    movel([0.144923, -1.275155, -2.596829, -0.840405, 1.570796, 1.715720],accel_mss,speed_ms,0,blend_radius_m)
    movel([0.144342, -1.274168, -2.597401, -0.840819, 1.570796, 1.715139],accel_mss,speed_ms,0,blend_radius_m)
    movel([0.143423, -1.273257, -2.597929, -0.841203, 1.570796, 1.714219],accel_mss,speed_ms,0,blend_radius_m)
    movel([0.142097, -1.272464, -2.598387, -0.841538, 1.570796, 1.712893],accel_mss,speed_ms,0,blend_radius_m)
    movel([0.140296, -1.271830, -2.598753, -0.841806, 1.570796, 1.711092],accel_mss,speed_ms,0,blend_radius_m)
    # Splitting Linear movement in 4 (instruction 536: MoveL 457)
    movel([0.138191, -1.271393, -2.599005, -0.841991, 1.570796, 1.708987],accel_mss,speed_ms,0,blend_radius_m)
    movel([0.136082, -1.270961, -2.599254, -0.842174, 1.570796, 1.706878],accel_mss,speed_ms,0,blend_radius_m)
    movel([0.133968, -1.270534, -2.599499, -0.842356, 1.570796, 1.704764],accel_mss,speed_ms,0,blend_radius_m)
    movel([0.131850, -1.270113, -2.599741, -0.842535, 1.570796, 1.702647],accel_mss,speed_ms,0,blend_radius_m)
    # Splitting Linear movement in 6 (instruction 537: MoveL 458)
    movel([0.129903, -1.269748, -2.599951, -0.842690, 1.570796, 1.700700],accel_mss,speed_ms,0,blend_radius_m)
    movel([0.127953, -1.269388, -2.600157, -0.842843, 1.570796, 1.698749],accel_mss,speed_ms,0,blend_radius_m)
    movel([0.125999, -1.269032, -2.600361, -0.842995, 1.570796, 1.696795],accel_mss,speed_ms,0,blend_radius_m)
    movel([0.124041, -1.268681, -2.600563, -0.843145, 1.570796, 1.694838],accel_mss,speed_ms,0,blend_radius_m)
    movel([0.122081, -1.268335, -2.600761, -0.843293, 1.570796, 1.692877],accel_mss,speed_ms,0,blend_radius_m)
    movel([0.120116, -1.267993, -2.600957, -0.843439, 1.570796, 1.690913],accel_mss,speed_ms,0,blend_radius_m)
    speed_ms = 0.005
    # Splitting Linear movement in 4 (instruction 539: MoveL 459)
    movel([0.120116, -1.265890, -2.599818, -0.846681, 1.570796, 1.690913],accel_mss,speed_ms,0,blend_radius_m)
    movel([0.120116, -1.263799, -2.598675, -0.849915, 1.570796, 1.690913],accel_mss,speed_ms,0,blend_radius_m)
    movel([0.120116, -1.261719, -2.597530, -0.853140, 1.570796, 1.690913],accel_mss,speed_ms,0,blend_radius_m)
    movel([0.120116, -1.259651, -2.596381, -0.856357, 1.570796, 1.690913],accel_mss,speed_ms,0,blend_radius_m)
    speed_ms = 0.040
    # Splitting Linear movement in 12 (instruction 541: MoveL 460)
    movel([0.118639, -1.261858, -2.595130, -0.855401, 1.570796, 1.689436],accel_mss,speed_ms,0,blend_radius_m)
    movel([0.117169, -1.264057, -2.593878, -0.854454, 1.570796, 1.687965],accel_mss,speed_ms,0,blend_radius_m)
    movel([0.115705, -1.266250, -2.592623, -0.853516, 1.570796, 1.686501],accel_mss,speed_ms,0,blend_radius_m)
    movel([0.114247, -1.268435, -2.591368, -0.852586, 1.570796, 1.685043],accel_mss,speed_ms,0,blend_radius_m)
    movel([0.112796, -1.270613, -2.590110, -0.851666, 1.570796, 1.683592],accel_mss,speed_ms,0,blend_radius_m)
    movel([0.111350, -1.272785, -2.588851, -0.850753, 1.570796, 1.682147],accel_mss,speed_ms,0,blend_radius_m)
    movel([0.109912, -1.274949, -2.587590, -0.849850, 1.570796, 1.680708],accel_mss,speed_ms,0,blend_radius_m)
    movel([0.108479, -1.277107, -2.586327, -0.848955, 1.570796, 1.679275],accel_mss,speed_ms,0,blend_radius_m)
    movel([0.107053, -1.279258, -2.585063, -0.848068, 1.570796, 1.677849],accel_mss,speed_ms,0,blend_radius_m)
    movel([0.105632, -1.281402, -2.583797, -0.847190, 1.570796, 1.676429],accel_mss,speed_ms,0,blend_radius_m)
    movel([0.104218, -1.283539, -2.582530, -0.846320, 1.570796, 1.675014],accel_mss,speed_ms,0,blend_radius_m)
    movel([0.102810, -1.285670, -2.581261, -0.845458, 1.570796, 1.673606],accel_mss,speed_ms,0,blend_radius_m)
    speed_ms = 0.005
    # Splitting Linear movement in 4 (instruction 543: MoveL 461)
    movel([0.102810, -1.287713, -2.582382, -0.842294, 1.570796, 1.673606],accel_mss,speed_ms,0,blend_radius_m)
    movel([0.102810, -1.289767, -2.583499, -0.839123, 1.570796, 1.673606],accel_mss,speed_ms,0,blend_radius_m)
    movel([0.102810, -1.291832, -2.584614, -0.835943, 1.570796, 1.673606],accel_mss,speed_ms,0,blend_radius_m)
    movel([0.102810, -1.293908, -2.585724, -0.832757, 1.570796, 1.673606],accel_mss,speed_ms,0,blend_radius_m)
    speed_ms = 0.035
    # Splitting Linear movement in 4 (instruction 545: MoveL 462)
    movel([0.104961, -1.293243, -2.586126, -0.833020, 1.570796, 1.675758],accel_mss,speed_ms,0,blend_radius_m)
    movel([0.107114, -1.292580, -2.586525, -0.833284, 1.570796, 1.677910],accel_mss,speed_ms,0,blend_radius_m)
    movel([0.109268, -1.291921, -2.586922, -0.833546, 1.570796, 1.680064],accel_mss,speed_ms,0,blend_radius_m)
    movel([0.111423, -1.291264, -2.587316, -0.833808, 1.570796, 1.682219],accel_mss,speed_ms,0,blend_radius_m)
    speed_ms = 0.005
    # Splitting Linear movement in 6 (instruction 547: MoveL 463)
    movel([0.111423, -1.289877, -2.586574, -0.835938, 1.570796, 1.682219],accel_mss,speed_ms,0,blend_radius_m)
    movel([0.111423, -1.288495, -2.585831, -0.838063, 1.570796, 1.682219],accel_mss,speed_ms,0,blend_radius_m)
    movel([0.111423, -1.287118, -2.585085, -0.840186, 1.570796, 1.682219],accel_mss,speed_ms,0,blend_radius_m)
    movel([0.111423, -1.285745, -2.584339, -0.842305, 1.570796, 1.682219],accel_mss,speed_ms,0,blend_radius_m)
    movel([0.111423, -1.284378, -2.583591, -0.844421, 1.570796, 1.682219],accel_mss,speed_ms,0,blend_radius_m)
    movel([0.111423, -1.283015, -2.582841, -0.846533, 1.570796, 1.682219],accel_mss,speed_ms,0,blend_radius_m)
    speed_ms = 0.040
    # Splitting Linear movement in 6 (instruction 549: MoveL 464)
    movel([0.113420, -1.282408, -2.583201, -0.846780, 1.570796, 1.684216],accel_mss,speed_ms,0,blend_radius_m)
    movel([0.115418, -1.281804, -2.583559, -0.847026, 1.570796, 1.686214],accel_mss,speed_ms,0,blend_radius_m)
    movel([0.117416, -1.281203, -2.583915, -0.847271, 1.570796, 1.688213],accel_mss,speed_ms,0,blend_radius_m)
    movel([0.119416, -1.280604, -2.584269, -0.847516, 1.570796, 1.690212],accel_mss,speed_ms,0,blend_radius_m)
    movel([0.121417, -1.280007, -2.584621, -0.847761, 1.570796, 1.692213],accel_mss,speed_ms,0,blend_radius_m)
    movel([0.123418, -1.279413, -2.584971, -0.848004, 1.570796, 1.694214],accel_mss,speed_ms,0,blend_radius_m)
    speed_ms = 0.005
    # Splitting Linear movement in 6 (instruction 551: MoveL 465)
    movel([0.123418, -1.280778, -2.585724, -0.845887, 1.570796, 1.694214],accel_mss,speed_ms,0,blend_radius_m)
    movel([0.123418, -1.282148, -2.586474, -0.843766, 1.570796, 1.694214],accel_mss,speed_ms,0,blend_radius_m)
    movel([0.123418, -1.283523, -2.587224, -0.841642, 1.570796, 1.694214],accel_mss,speed_ms,0,blend_radius_m)
    movel([0.123418, -1.284903, -2.587971, -0.839515, 1.570796, 1.694214],accel_mss,speed_ms,0,blend_radius_m)
    movel([0.123418, -1.286288, -2.588717, -0.837384, 1.570796, 1.694214],accel_mss,speed_ms,0,blend_radius_m)
    movel([0.123418, -1.287678, -2.589462, -0.835249, 1.570796, 1.694214],accel_mss,speed_ms,0,blend_radius_m)
    speed_ms = 0.035
    # Splitting Linear movement in 4 (instruction 553: MoveL 466)
    movel([0.125386, -1.287119, -2.589795, -0.835475, 1.570796, 1.696182],accel_mss,speed_ms,0,blend_radius_m)
    movel([0.127354, -1.286563, -2.590126, -0.835700, 1.570796, 1.698151],accel_mss,speed_ms,0,blend_radius_m)
    movel([0.129323, -1.286009, -2.590455, -0.835925, 1.570796, 1.700120],accel_mss,speed_ms,0,blend_radius_m)
    movel([0.131293, -1.285459, -2.590782, -0.836149, 1.570796, 1.702090],accel_mss,speed_ms,0,blend_radius_m)
    movel([0.133014, -1.284863, -2.591135, -0.836391, 1.570796, 1.703811],accel_mss,speed_ms,0,blend_radius_m)
    movel([0.134155, -1.284224, -2.591513, -0.836652, 1.570796, 1.704951],accel_mss,speed_ms,0,blend_radius_m)
    movel([0.135046, -1.283460, -2.591965, -0.836964, 1.570796, 1.705842],accel_mss,speed_ms,0,blend_radius_m)
    movel([0.135680, -1.282694, -2.592417, -0.837278, 1.570796, 1.706476],accel_mss,speed_ms,0,blend_radius_m)
    movel([0.136054, -1.282045, -2.592800, -0.837544, 1.570796, 1.706850],accel_mss,speed_ms,0,blend_radius_m)
    movel([0.136254, -1.281407, -2.593175, -0.837807, 1.570796, 1.707050],accel_mss,speed_ms,0,blend_radius_m)
    movel([0.136336, -1.280413, -2.593759, -0.838217, 1.570796, 1.707133],accel_mss,speed_ms,0,blend_radius_m)
    movel([0.136227, -1.279892, -2.594065, -0.838432, 1.570796, 1.707023],accel_mss,speed_ms,0,blend_radius_m)
    movel([0.135967, -1.279413, -2.594346, -0.838630, 1.570796, 1.706763],accel_mss,speed_ms,0,blend_radius_m)
    movel([0.135513, -1.279021, -2.594575, -0.838792, 1.570796, 1.706310],accel_mss,speed_ms,0,blend_radius_m)
    movel([0.134824, -1.278762, -2.594727, -0.838900, 1.570796, 1.705620],accel_mss,speed_ms,0,blend_radius_m)
    # Splitting Linear movement in 6 (instruction 565: MoveL 478)
    movel([0.132749, -1.278413, -2.594931, -0.839045, 1.570796, 1.703546],accel_mss,speed_ms,0,blend_radius_m)
    movel([0.130671, -1.278069, -2.595132, -0.839188, 1.570796, 1.701467],accel_mss,speed_ms,0,blend_radius_m)
    movel([0.128589, -1.277730, -2.595330, -0.839329, 1.570796, 1.699385],accel_mss,speed_ms,0,blend_radius_m)
    movel([0.126503, -1.277396, -2.595525, -0.839468, 1.570796, 1.697299],accel_mss,speed_ms,0,blend_radius_m)
    movel([0.124413, -1.277068, -2.595716, -0.839605, 1.570796, 1.695210],accel_mss,speed_ms,0,blend_radius_m)
    movel([0.122320, -1.276744, -2.595905, -0.839740, 1.570796, 1.693117],accel_mss,speed_ms,0,blend_radius_m)
    # Splitting Linear movement in 8 (instruction 566: MoveL 479)
    movel([0.122076, -1.278708, -2.594758, -0.838922, 1.570796, 1.692872],accel_mss,speed_ms,0,blend_radius_m)
    movel([0.121832, -1.280667, -2.593610, -0.838112, 1.570796, 1.692628],accel_mss,speed_ms,0,blend_radius_m)
    movel([0.121589, -1.282620, -2.592461, -0.837308, 1.570796, 1.692386],accel_mss,speed_ms,0,blend_radius_m)
    movel([0.121348, -1.284567, -2.591310, -0.836512, 1.570796, 1.692144],accel_mss,speed_ms,0,blend_radius_m)
    movel([0.121107, -1.286509, -2.590158, -0.835722, 1.570796, 1.691903],accel_mss,speed_ms,0,blend_radius_m)
    movel([0.120868, -1.288446, -2.589004, -0.834939, 1.570796, 1.691664],accel_mss,speed_ms,0,blend_radius_m)
    movel([0.120629, -1.290377, -2.587849, -0.834163, 1.570796, 1.691426],accel_mss,speed_ms,0,blend_radius_m)
    movel([0.120392, -1.292303, -2.586692, -0.833394, 1.570796, 1.691188],accel_mss,speed_ms,0,blend_radius_m)
    speed_ms = 0.005
    # Splitting Linear movement in 4 (instruction 568: MoveL 480)
    movel([0.120392, -1.290225, -2.585579, -0.836584, 1.570796, 1.691188],accel_mss,speed_ms,0,blend_radius_m)
    movel([0.120392, -1.288159, -2.584463, -0.839767, 1.570796, 1.691188],accel_mss,speed_ms,0,blend_radius_m)
    movel([0.120392, -1.286103, -2.583344, -0.842942, 1.570796, 1.691188],accel_mss,speed_ms,0,blend_radius_m)
    movel([0.120392, -1.284058, -2.582221, -0.846110, 1.570796, 1.691188],accel_mss,speed_ms,0,blend_radius_m)
    speed_ms = 0.040
    # Splitting Linear movement in 12 (instruction 570: MoveL 481)
    movel([0.119907, -1.286179, -2.580956, -0.845253, 1.570796, 1.690703],accel_mss,speed_ms,0,blend_radius_m)
    movel([0.119424, -1.288294, -2.579690, -0.844405, 1.570796, 1.690220],accel_mss,speed_ms,0,blend_radius_m)
    movel([0.118943, -1.290401, -2.578422, -0.843565, 1.570796, 1.689739],accel_mss,speed_ms,0,blend_radius_m)
    movel([0.118465, -1.292503, -2.577153, -0.842733, 1.570796, 1.689261],accel_mss,speed_ms,0,blend_radius_m)
    movel([0.117988, -1.294598, -2.575882, -0.841909, 1.570796, 1.688785],accel_mss,speed_ms,0,blend_radius_m)
    movel([0.117514, -1.296686, -2.574609, -0.841093, 1.570796, 1.688311],accel_mss,speed_ms,0,blend_radius_m)
    movel([0.117042, -1.298768, -2.573335, -0.840285, 1.570796, 1.687839],accel_mss,speed_ms,0,blend_radius_m)
    movel([0.116573, -1.300844, -2.572060, -0.839485, 1.570796, 1.687369],accel_mss,speed_ms,0,blend_radius_m)
    movel([0.116105, -1.302914, -2.570782, -0.838693, 1.570796, 1.686901],accel_mss,speed_ms,0,blend_radius_m)
    movel([0.115640, -1.304977, -2.569504, -0.837908, 1.570796, 1.686436],accel_mss,speed_ms,0,blend_radius_m)
    movel([0.115176, -1.307034, -2.568224, -0.837131, 1.570796, 1.685973],accel_mss,speed_ms,0,blend_radius_m)
    movel([0.114715, -1.309085, -2.566942, -0.836362, 1.570796, 1.685512],accel_mss,speed_ms,0,blend_radius_m)
    speed_ms = 0.005
    # Splitting Linear movement in 6 (instruction 572: MoveL 482)
    movel([0.114715, -1.310429, -2.567673, -0.834287, 1.570796, 1.685512],accel_mss,speed_ms,0,blend_radius_m)
    movel([0.114715, -1.311778, -2.568403, -0.832208, 1.570796, 1.685512],accel_mss,speed_ms,0,blend_radius_m)
    movel([0.114715, -1.313131, -2.569131, -0.830127, 1.570796, 1.685512],accel_mss,speed_ms,0,blend_radius_m)
    movel([0.114715, -1.314489, -2.569857, -0.828042, 1.570796, 1.685512],accel_mss,speed_ms,0,blend_radius_m)
    movel([0.114715, -1.315852, -2.570582, -0.825955, 1.570796, 1.685512],accel_mss,speed_ms,0,blend_radius_m)
    movel([0.114715, -1.317219, -2.571306, -0.823864, 1.570796, 1.685512],accel_mss,speed_ms,0,blend_radius_m)
    speed_ms = 0.035
    movel([0.113872, -1.317605, -2.571061, -0.823723, 1.570796, 1.684668],accel_mss,speed_ms,0,blend_radius_m)
    movel([0.113052, -1.317884, -2.570884, -0.823621, 1.570796, 1.683848],accel_mss,speed_ms,0,blend_radius_m)
    movel([0.111543, -1.318120, -2.570734, -0.823534, 1.570796, 1.682339],accel_mss,speed_ms,0,blend_radius_m)
    movel([0.110880, -1.318079, -2.570761, -0.823550, 1.570796, 1.681676],accel_mss,speed_ms,0,blend_radius_m)
    movel([0.109799, -1.317678, -2.571015, -0.823696, 1.570796, 1.680595],accel_mss,speed_ms,0,blend_radius_m)
    movel([0.109406, -1.317320, -2.571242, -0.823827, 1.570796, 1.680202],accel_mss,speed_ms,0,blend_radius_m)
    movel([0.108993, -1.316375, -2.571840, -0.824174, 1.570796, 1.679790],accel_mss,speed_ms,0,blend_radius_m)
    movel([0.108987, -1.315364, -2.572479, -0.824546, 1.570796, 1.679783],accel_mss,speed_ms,0,blend_radius_m)
    movel([0.109341, -1.314017, -2.573327, -0.825045, 1.570796, 1.680137],accel_mss,speed_ms,0,blend_radius_m)
    movel([0.109909, -1.312888, -2.574037, -0.825464, 1.570796, 1.680705],accel_mss,speed_ms,0,blend_radius_m)
    movel([0.110621, -1.311896, -2.574659, -0.825834, 1.570796, 1.681417],accel_mss,speed_ms,0,blend_radius_m)
    movel([0.111393, -1.311055, -2.575186, -0.826148, 1.570796, 1.682189],accel_mss,speed_ms,0,blend_radius_m)
    movel([0.112144, -1.310376, -2.575611, -0.826403, 1.570796, 1.682940],accel_mss,speed_ms,0,blend_radius_m)
    movel([0.114992, -1.307950, -2.577122, -0.827317, 1.570796, 1.685788],accel_mss,speed_ms,0,blend_radius_m)
    movel([0.116059, -1.306889, -2.577780, -0.827719, 1.570796, 1.686856],accel_mss,speed_ms,0,blend_radius_m)
    movel([0.117029, -1.305645, -2.578551, -0.828193, 1.570796, 1.687826],accel_mss,speed_ms,0,blend_radius_m)
    movel([0.117834, -1.304414, -2.579312, -0.828663, 1.570796, 1.688630],accel_mss,speed_ms,0,blend_radius_m)
    movel([0.118394, -1.303386, -2.579945, -0.829058, 1.570796, 1.689190],accel_mss,speed_ms,0,blend_radius_m)
    movel([0.118876, -1.302219, -2.580663, -0.829507, 1.570796, 1.689672],accel_mss,speed_ms,0,blend_radius_m)
    movel([0.119170, -1.301159, -2.581313, -0.829917, 1.570796, 1.689966],accel_mss,speed_ms,0,blend_radius_m)
    movel([0.119460, -1.299307, -2.582446, -0.830636, 1.570796, 1.690257],accel_mss,speed_ms,0,blend_radius_m)
    speed_ms = 0.005
    # Splitting Linear movement in 6 (instruction 596: MoveL 504)
    movel([0.119460, -1.297926, -2.581710, -0.832753, 1.570796, 1.690257],accel_mss,speed_ms,0,blend_radius_m)
    movel([0.119460, -1.296550, -2.580972, -0.834867, 1.570796, 1.690257],accel_mss,speed_ms,0,blend_radius_m)
    movel([0.119460, -1.295178, -2.580233, -0.836978, 1.570796, 1.690257],accel_mss,speed_ms,0,blend_radius_m)
    movel([0.119460, -1.293811, -2.579492, -0.839086, 1.570796, 1.690257],accel_mss,speed_ms,0,blend_radius_m)
    movel([0.119460, -1.292450, -2.578749, -0.841190, 1.570796, 1.690257],accel_mss,speed_ms,0,blend_radius_m)
    movel([0.119460, -1.291092, -2.578005, -0.843291, 1.570796, 1.690257],accel_mss,speed_ms,0,blend_radius_m)
    speed_ms = 0.040
    # Splitting Linear movement in 4 (instruction 598: MoveL 505)
    movel([0.117830, -1.291504, -2.577757, -0.843128, 1.570796, 1.688627],accel_mss,speed_ms,0,blend_radius_m)
    movel([0.116201, -1.291917, -2.577507, -0.842965, 1.570796, 1.686997],accel_mss,speed_ms,0,blend_radius_m)
    movel([0.114572, -1.292332, -2.577256, -0.842801, 1.570796, 1.685368],accel_mss,speed_ms,0,blend_radius_m)
    movel([0.112943, -1.292749, -2.577004, -0.842636, 1.570796, 1.683739],accel_mss,speed_ms,0,blend_radius_m)
    speed_ms = 0.005
    # Splitting Linear movement in 6 (instruction 600: MoveL 506)
    movel([0.112943, -1.294105, -2.577746, -0.840537, 1.570796, 1.683739],accel_mss,speed_ms,0,blend_radius_m)
    movel([0.112943, -1.295466, -2.578488, -0.838435, 1.570796, 1.683739],accel_mss,speed_ms,0,blend_radius_m)
    movel([0.112943, -1.296831, -2.579227, -0.836330, 1.570796, 1.683739],accel_mss,speed_ms,0,blend_radius_m)
    movel([0.112943, -1.298202, -2.579965, -0.834222, 1.570796, 1.683739],accel_mss,speed_ms,0,blend_radius_m)
    movel([0.112943, -1.299577, -2.580702, -0.832110, 1.570796, 1.683739],accel_mss,speed_ms,0,blend_radius_m)
    movel([0.112943, -1.300957, -2.581437, -0.829995, 1.570796, 1.683739],accel_mss,speed_ms,0,blend_radius_m)
    speed_ms = 0.035
    movel([0.112634, -1.302487, -2.580498, -0.829404, 1.570796, 1.683431],accel_mss,speed_ms,0,blend_radius_m)
    movel([0.112220, -1.303581, -2.579825, -0.828983, 1.570796, 1.683016],accel_mss,speed_ms,0,blend_radius_m)
    movel([0.111539, -1.304692, -2.579140, -0.828557, 1.570796, 1.682335],accel_mss,speed_ms,0,blend_radius_m)
    movel([0.110449, -1.305905, -2.578390, -0.828094, 1.570796, 1.681246],accel_mss,speed_ms,0,blend_radius_m)
    movel([0.109369, -1.306856, -2.577801, -0.827732, 1.570796, 1.680165],accel_mss,speed_ms,0,blend_radius_m)
    movel([0.107828, -1.307928, -2.577136, -0.827326, 1.570796, 1.678624],accel_mss,speed_ms,0,blend_radius_m)
    speed_ms = 0.005
    # Splitting Linear movement in 6 (instruction 609: MoveL 513)
    movel([0.107828, -1.306553, -2.576405, -0.829430, 1.570796, 1.678624],accel_mss,speed_ms,0,blend_radius_m)
    movel([0.107828, -1.305184, -2.575674, -0.831532, 1.570796, 1.678624],accel_mss,speed_ms,0,blend_radius_m)
    movel([0.107828, -1.303819, -2.574940, -0.833630, 1.570796, 1.678624],accel_mss,speed_ms,0,blend_radius_m)
    movel([0.107828, -1.302458, -2.574206, -0.835725, 1.570796, 1.678624],accel_mss,speed_ms,0,blend_radius_m)
    movel([0.107828, -1.301103, -2.573470, -0.837817, 1.570796, 1.678624],accel_mss,speed_ms,0,blend_radius_m)
    movel([0.107828, -1.299752, -2.572732, -0.839906, 1.570796, 1.678624],accel_mss,speed_ms,0,blend_radius_m)
    speed_ms = 0.040
    # Splitting Linear movement in 6 (instruction 611: MoveL 514)
    movel([0.108730, -1.297552, -2.574080, -0.840757, 1.570796, 1.679526],accel_mss,speed_ms,0,blend_radius_m)
    movel([0.109636, -1.295346, -2.575427, -0.841616, 1.570796, 1.680432],accel_mss,speed_ms,0,blend_radius_m)
    movel([0.110546, -1.293132, -2.576772, -0.842485, 1.570796, 1.681343],accel_mss,speed_ms,0,blend_radius_m)
    movel([0.111461, -1.290911, -2.578115, -0.843363, 1.570796, 1.682257],accel_mss,speed_ms,0,blend_radius_m)
    movel([0.112380, -1.288682, -2.579457, -0.844250, 1.570796, 1.683176],accel_mss,speed_ms,0,blend_radius_m)
    movel([0.113304, -1.286446, -2.580797, -0.845146, 1.570796, 1.684100],accel_mss,speed_ms,0,blend_radius_m)
    speed_ms = 0.005
    # Splitting Linear movement in 4 (instruction 613: MoveL 515)
    movel([0.113304, -1.288488, -2.581917, -0.841984, 1.570796, 1.684100],accel_mss,speed_ms,0,blend_radius_m)
    movel([0.113304, -1.290541, -2.583034, -0.838813, 1.570796, 1.684100],accel_mss,speed_ms,0,blend_radius_m)
    movel([0.113304, -1.292606, -2.584148, -0.835636, 1.570796, 1.684100],accel_mss,speed_ms,0,blend_radius_m)
    movel([0.113304, -1.294681, -2.585258, -0.832451, 1.570796, 1.684100],accel_mss,speed_ms,0,blend_radius_m)
    speed_ms = 0.035
    # Splitting Linear movement in 10 (instruction 615: MoveL 516)
    movel([0.113551, -1.292716, -2.586443, -0.833230, 1.570796, 1.684348],accel_mss,speed_ms,0,blend_radius_m)
    movel([0.113800, -1.290745, -2.587628, -0.834016, 1.570796, 1.684596],accel_mss,speed_ms,0,blend_radius_m)
    movel([0.114050, -1.288769, -2.588811, -0.834809, 1.570796, 1.684846],accel_mss,speed_ms,0,blend_radius_m)
    movel([0.114301, -1.286787, -2.589992, -0.835609, 1.570796, 1.685097],accel_mss,speed_ms,0,blend_radius_m)
    movel([0.114553, -1.284800, -2.591172, -0.836417, 1.570796, 1.685349],accel_mss,speed_ms,0,blend_radius_m)
    movel([0.114806, -1.282807, -2.592350, -0.837232, 1.570796, 1.685603],accel_mss,speed_ms,0,blend_radius_m)
    movel([0.115061, -1.280808, -2.593527, -0.838053, 1.570796, 1.685857],accel_mss,speed_ms,0,blend_radius_m)
    movel([0.115316, -1.278804, -2.594703, -0.838883, 1.570796, 1.686113],accel_mss,speed_ms,0,blend_radius_m)
    movel([0.115573, -1.276793, -2.595876, -0.839719, 1.570796, 1.686370],accel_mss,speed_ms,0,blend_radius_m)
    movel([0.115831, -1.274777, -2.597048, -0.840563, 1.570796, 1.686627],accel_mss,speed_ms,0,blend_radius_m)
    speed_ms = 0.005
    # Splitting Linear movement in 6 (instruction 617: MoveL 517)
    movel([0.115831, -1.273379, -2.596294, -0.842716, 1.570796, 1.686627],accel_mss,speed_ms,0,blend_radius_m)
    movel([0.115831, -1.271985, -2.595539, -0.844865, 1.570796, 1.686627],accel_mss,speed_ms,0,blend_radius_m)
    movel([0.115831, -1.270596, -2.594782, -0.847011, 1.570796, 1.686627],accel_mss,speed_ms,0,blend_radius_m)
    movel([0.115831, -1.269213, -2.594023, -0.849153, 1.570796, 1.686627],accel_mss,speed_ms,0,blend_radius_m)
    movel([0.115831, -1.267835, -2.593263, -0.851291, 1.570796, 1.686627],accel_mss,speed_ms,0,blend_radius_m)
    movel([0.115831, -1.266461, -2.592502, -0.853426, 1.570796, 1.686627],accel_mss,speed_ms,0,blend_radius_m)
    speed_ms = 0.040
    # Splitting Linear movement in 14 (instruction 619: MoveL 518)
    movel([0.115694, -1.264402, -2.593681, -0.854307, 1.570796, 1.686491],accel_mss,speed_ms,0,blend_radius_m)
    movel([0.115557, -1.262336, -2.594858, -0.855195, 1.570796, 1.686354],accel_mss,speed_ms,0,blend_radius_m)
    movel([0.115419, -1.260266, -2.596033, -0.856090, 1.570796, 1.686216],accel_mss,speed_ms,0,blend_radius_m)
    movel([0.115281, -1.258190, -2.597205, -0.856993, 1.570796, 1.686077],accel_mss,speed_ms,0,blend_radius_m)
    movel([0.115141, -1.256109, -2.598376, -0.857904, 1.570796, 1.685938],accel_mss,speed_ms,0,blend_radius_m)
    movel([0.115001, -1.254023, -2.599545, -0.858821, 1.570796, 1.685798],accel_mss,speed_ms,0,blend_radius_m)
    movel([0.114861, -1.251931, -2.600711, -0.859747, 1.570796, 1.685657],accel_mss,speed_ms,0,blend_radius_m)
    movel([0.114719, -1.249834, -2.601875, -0.860680, 1.570796, 1.685515],accel_mss,speed_ms,0,blend_radius_m)
    movel([0.114577, -1.247731, -2.603037, -0.861621, 1.570796, 1.685373],accel_mss,speed_ms,0,blend_radius_m)
    movel([0.114434, -1.245623, -2.604197, -0.862569, 1.570796, 1.685231],accel_mss,speed_ms,0,blend_radius_m)
    movel([0.114291, -1.243509, -2.605355, -0.863525, 1.570796, 1.685087],accel_mss,speed_ms,0,blend_radius_m)
    movel([0.114147, -1.241390, -2.606511, -0.864488, 1.570796, 1.684943],accel_mss,speed_ms,0,blend_radius_m)
    movel([0.114002, -1.239265, -2.607664, -0.865460, 1.570796, 1.684798],accel_mss,speed_ms,0,blend_radius_m)
    movel([0.113856, -1.237135, -2.608815, -0.866439, 1.570796, 1.684652],accel_mss,speed_ms,0,blend_radius_m)
    speed_ms = 0.005
    # Splitting Linear movement in 6 (instruction 621: MoveL 519)
    movel([0.113856, -1.238525, -2.609598, -0.864266, 1.570796, 1.684652],accel_mss,speed_ms,0,blend_radius_m)
    movel([0.113856, -1.239920, -2.610379, -0.862090, 1.570796, 1.684652],accel_mss,speed_ms,0,blend_radius_m)
    movel([0.113856, -1.241321, -2.611158, -0.859909, 1.570796, 1.684652],accel_mss,speed_ms,0,blend_radius_m)
    movel([0.113856, -1.242728, -2.611937, -0.857725, 1.570796, 1.684652],accel_mss,speed_ms,0,blend_radius_m)
    movel([0.113856, -1.244139, -2.612713, -0.855537, 1.570796, 1.684652],accel_mss,speed_ms,0,blend_radius_m)
    movel([0.113856, -1.245557, -2.613488, -0.853344, 1.570796, 1.684652],accel_mss,speed_ms,0,blend_radius_m)
    speed_ms = 0.035
    movel([0.112072, -1.247704, -2.612315, -0.852371, 1.570796, 1.682869],accel_mss,speed_ms,0,blend_radius_m)
    movel([0.111082, -1.249111, -2.611543, -0.851735, 1.570796, 1.681878],accel_mss,speed_ms,0,blend_radius_m)
    movel([0.110109, -1.250720, -2.610657, -0.851012, 1.570796, 1.680905],accel_mss,speed_ms,0,blend_radius_m)
    movel([0.108800, -1.253463, -2.609140, -0.849786, 1.570796, 1.679596],accel_mss,speed_ms,0,blend_radius_m)
    movel([0.108042, -1.255743, -2.607873, -0.848773, 1.570796, 1.678838],accel_mss,speed_ms,0,blend_radius_m)
    movel([0.107678, -1.257501, -2.606891, -0.847997, 1.570796, 1.678475],accel_mss,speed_ms,0,blend_radius_m)
    movel([0.107571, -1.259744, -2.605634, -0.847012, 1.570796, 1.678367],accel_mss,speed_ms,0,blend_radius_m)
    movel([0.107728, -1.261120, -2.604859, -0.846410, 1.570796, 1.678524],accel_mss,speed_ms,0,blend_radius_m)
    movel([0.108137, -1.262661, -2.603989, -0.845739, 1.570796, 1.678933],accel_mss,speed_ms,0,blend_radius_m)
    movel([0.108894, -1.264225, -2.603103, -0.845061, 1.570796, 1.679690],accel_mss,speed_ms,0,blend_radius_m)
    movel([0.109910, -1.265454, -2.602405, -0.844530, 1.570796, 1.680707],accel_mss,speed_ms,0,blend_radius_m)
    movel([0.110987, -1.266309, -2.601918, -0.844162, 1.570796, 1.681784],accel_mss,speed_ms,0,blend_radius_m)
    movel([0.112503, -1.267102, -2.601466, -0.843821, 1.570796, 1.683299],accel_mss,speed_ms,0,blend_radius_m)
    movel([0.114619, -1.267684, -2.601133, -0.843572, 1.570796, 1.685415],accel_mss,speed_ms,0,blend_radius_m)
    movel([0.116412, -1.267846, -2.601040, -0.843502, 1.570796, 1.687208],accel_mss,speed_ms,0,blend_radius_m)
    speed_ms = 0.005
    # Splitting Linear movement in 22 (instruction 639: MoveL 535)
    movel([0.116412, -1.265934, -2.600005, -0.846450, 1.570796, 1.687208],accel_mss,speed_ms,0,blend_radius_m)
    movel([0.116412, -1.264031, -2.598967, -0.849391, 1.570796, 1.687208],accel_mss,speed_ms,0,blend_radius_m)
    movel([0.116412, -1.262138, -2.597926, -0.852325, 1.570796, 1.687208],accel_mss,speed_ms,0,blend_radius_m)
    movel([0.116412, -1.260254, -2.596882, -0.855252, 1.570796, 1.687208],accel_mss,speed_ms,0,blend_radius_m)
    movel([0.116412, -1.258380, -2.595836, -0.858173, 1.570796, 1.687208],accel_mss,speed_ms,0,blend_radius_m)
    movel([0.116412, -1.256516, -2.594787, -0.861086, 1.570796, 1.687208],accel_mss,speed_ms,0,blend_radius_m)
    movel([0.116412, -1.254661, -2.593735, -0.863993, 1.570796, 1.687208],accel_mss,speed_ms,0,blend_radius_m)
    movel([0.116412, -1.252815, -2.592680, -0.866893, 1.570796, 1.687208],accel_mss,speed_ms,0,blend_radius_m)
    movel([0.116412, -1.250979, -2.591623, -0.869787, 1.570796, 1.687208],accel_mss,speed_ms,0,blend_radius_m)
    movel([0.116412, -1.249153, -2.590563, -0.872673, 1.570796, 1.687208],accel_mss,speed_ms,0,blend_radius_m)
    movel([0.116412, -1.247336, -2.589500, -0.875553, 1.570796, 1.687208],accel_mss,speed_ms,0,blend_radius_m)
    movel([0.116412, -1.245528, -2.588435, -0.878426, 1.570796, 1.687208],accel_mss,speed_ms,0,blend_radius_m)
    movel([0.116412, -1.243729, -2.587367, -0.881293, 1.570796, 1.687208],accel_mss,speed_ms,0,blend_radius_m)
    movel([0.116412, -1.241940, -2.586296, -0.884153, 1.570796, 1.687208],accel_mss,speed_ms,0,blend_radius_m)
    movel([0.116412, -1.240160, -2.585223, -0.887006, 1.570796, 1.687208],accel_mss,speed_ms,0,blend_radius_m)
    movel([0.116412, -1.238390, -2.584147, -0.889852, 1.570796, 1.687208],accel_mss,speed_ms,0,blend_radius_m)
    movel([0.116412, -1.236629, -2.583068, -0.892692, 1.570796, 1.687208],accel_mss,speed_ms,0,blend_radius_m)
    movel([0.116412, -1.234876, -2.581987, -0.895525, 1.570796, 1.687208],accel_mss,speed_ms,0,blend_radius_m)
    movel([0.116412, -1.233134, -2.580904, -0.898352, 1.570796, 1.687208],accel_mss,speed_ms,0,blend_radius_m)
    movel([0.116412, -1.231400, -2.579817, -0.901172, 1.570796, 1.687208],accel_mss,speed_ms,0,blend_radius_m)
    movel([0.116412, -1.229675, -2.578729, -0.903985, 1.570796, 1.687208],accel_mss,speed_ms,0,blend_radius_m)
    movel([0.116412, -1.227960, -2.577637, -0.906792, 1.570796, 1.687208],accel_mss,speed_ms,0,blend_radius_m)
    speed_ms = 1.000
    movel([0.116412, -1.227960, -2.577637, -0.906792, 1.570796, 1.687208],accel_mss,speed_ms,0,blend_radius_m)
    # Splitting Linear movement in 32 (instruction 642: MoveL 537)
    movel([0.116412, -1.226200, -2.576509, -0.909680, 1.570796, 1.687208],accel_mss,speed_ms,0,blend_radius_m)
    movel([0.116412, -1.224450, -2.575378, -0.912560, 1.570796, 1.687208],accel_mss,speed_ms,0,blend_radius_m)
    movel([0.116412, -1.222710, -2.574245, -0.915434, 1.570796, 1.687208],accel_mss,speed_ms,0,blend_radius_m)
    movel([0.116412, -1.220979, -2.573109, -0.918301, 1.570796, 1.687208],accel_mss,speed_ms,0,blend_radius_m)
    movel([0.116412, -1.219258, -2.571970, -0.921161, 1.570796, 1.687208],accel_mss,speed_ms,0,blend_radius_m)
    movel([0.116412, -1.217546, -2.570829, -0.924014, 1.570796, 1.687208],accel_mss,speed_ms,0,blend_radius_m)
    movel([0.116412, -1.215844, -2.569685, -0.926860, 1.570796, 1.687208],accel_mss,speed_ms,0,blend_radius_m)
    movel([0.116412, -1.214151, -2.568538, -0.929699, 1.570796, 1.687208],accel_mss,speed_ms,0,blend_radius_m)
    movel([0.116412, -1.212468, -2.567389, -0.932532, 1.570796, 1.687208],accel_mss,speed_ms,0,blend_radius_m)
    movel([0.116412, -1.210794, -2.566238, -0.935358, 1.570796, 1.687208],accel_mss,speed_ms,0,blend_radius_m)
    movel([0.116412, -1.209129, -2.565083, -0.938176, 1.570796, 1.687208],accel_mss,speed_ms,0,blend_radius_m)
    movel([0.116412, -1.207474, -2.563926, -0.940989, 1.570796, 1.687208],accel_mss,speed_ms,0,blend_radius_m)
    movel([0.116412, -1.205828, -2.562767, -0.943794, 1.570796, 1.687208],accel_mss,speed_ms,0,blend_radius_m)
    movel([0.116412, -1.204191, -2.561605, -0.946593, 1.570796, 1.687208],accel_mss,speed_ms,0,blend_radius_m)
    movel([0.116412, -1.202564, -2.560441, -0.949385, 1.570796, 1.687208],accel_mss,speed_ms,0,blend_radius_m)
    movel([0.116412, -1.200945, -2.559274, -0.952170, 1.570796, 1.687208],accel_mss,speed_ms,0,blend_radius_m)
    movel([0.116412, -1.199336, -2.558104, -0.954948, 1.570796, 1.687208],accel_mss,speed_ms,0,blend_radius_m)
    movel([0.116412, -1.197736, -2.556932, -0.957720, 1.570796, 1.687208],accel_mss,speed_ms,0,blend_radius_m)
    movel([0.116412, -1.196145, -2.555758, -0.960486, 1.570796, 1.687208],accel_mss,speed_ms,0,blend_radius_m)
    movel([0.116412, -1.194564, -2.554581, -0.963244, 1.570796, 1.687208],accel_mss,speed_ms,0,blend_radius_m)
    movel([0.116412, -1.192991, -2.553402, -0.965996, 1.570796, 1.687208],accel_mss,speed_ms,0,blend_radius_m)
    movel([0.116412, -1.191427, -2.552220, -0.968742, 1.570796, 1.687208],accel_mss,speed_ms,0,blend_radius_m)
    movel([0.116412, -1.189872, -2.551036, -0.971481, 1.570796, 1.687208],accel_mss,speed_ms,0,blend_radius_m)
    movel([0.116412, -1.188326, -2.549849, -0.974213, 1.570796, 1.687208],accel_mss,speed_ms,0,blend_radius_m)
    movel([0.116412, -1.186790, -2.548661, -0.976939, 1.570796, 1.687208],accel_mss,speed_ms,0,blend_radius_m)
    movel([0.116412, -1.185262, -2.547469, -0.979658, 1.570796, 1.687208],accel_mss,speed_ms,0,blend_radius_m)
    movel([0.116412, -1.183742, -2.546275, -0.982371, 1.570796, 1.687208],accel_mss,speed_ms,0,blend_radius_m)
    movel([0.116412, -1.182232, -2.545079, -0.985078, 1.570796, 1.687208],accel_mss,speed_ms,0,blend_radius_m)
    movel([0.116412, -1.180730, -2.543881, -0.987778, 1.570796, 1.687208],accel_mss,speed_ms,0,blend_radius_m)
    movel([0.116412, -1.179238, -2.542680, -0.990471, 1.570796, 1.687208],accel_mss,speed_ms,0,blend_radius_m)
    movel([0.116412, -1.177754, -2.541477, -0.993158, 1.570796, 1.687208],accel_mss,speed_ms,0,blend_radius_m)
    movel([0.116412, -1.176278, -2.540271, -0.995839, 1.570796, 1.687208],accel_mss,speed_ms,0,blend_radius_m)
    # End of main program
  end

  Machining1()
end
